PROGRAM MAIN
VAR
	bInit	:BOOL;
END_VAR

P01_AxesControl();

END_PROGRAM

(* stored: Version 1.1.0.1, ProductVersion 3.1.4022.18
   POU MAIN: Id {5e903faa-f943-4e28-a98c-cbe6f1c42525}, SpecialFunc None *)
